(* Logix 5000 project; controller Drives_Line1 1756-L72 rev 20.13; software revision 20.04; part 14 of 21 *)
(* tags used below, declared in another part *)
   zEntry_Accu_MaxAccDec : REAL;
   zEntry_Accu_SpdRegMax : REAL;
   zEntry_Accu_SpdRegMin : REAL;
   Bridle_01 : UDT_Bridle_3M;
   Bridle_02 : UDT_Bridle_2M;
   Bridle_03 : UDT_Bridle_2M;
   Entry_Accu : UDT_Entry_Accu;
   EntryCtrl : UDT_Control_Zone;
   In_Commands : UDT_Commands;
   In_Config : UDT_Config;
   In_Setpoints : UDT_Setpoints;
   LineCmd : UDT_Commands_Line;
   LineCtrl : UDT_Control_Line;
   Out_Feedbacks : UDT_Fdbks;
   Out_Status : UDT_Status;
   TestConfig_Entry_Accu : UDT_Config_Accu;
   TM1 : UDT_TM;
   TM2 : UDT_TM;
   zConfigFromMaster : BOOL;
   zExit_Accu_NrOfCyl : DINT;
(* P16_Entry_Accu, continued *)

ROUTINE R12_DriveRef   (* function block diagram *)
   SHEET 1   // Speed reference selection
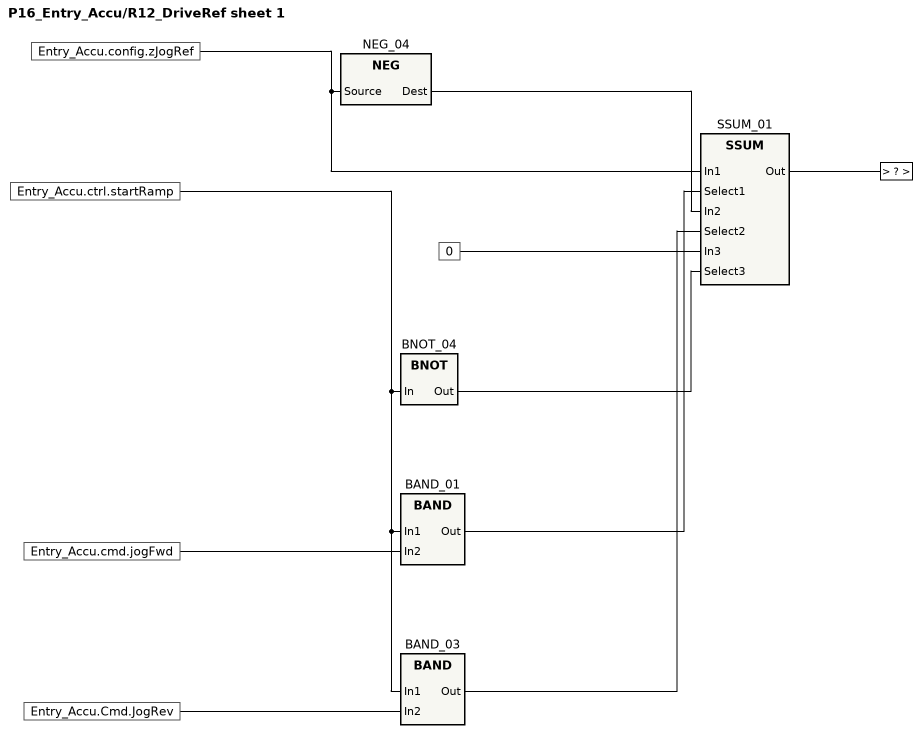
   NEG_04 : NEG(Source := Entry_Accu.config.zJogRef);
   BNOT_04 : BNOT(In := Entry_Accu.ctrl.startRamp);
   BAND_01 : BAND(In1 := Entry_Accu.ctrl.startRamp, In2 := Entry_Accu.cmd.jogFwd);
   BAND_03 : BAND(In1 := Entry_Accu.ctrl.startRamp, In2 := Entry_Accu.Cmd.JogRev);
   SSUM_01 : SSUM(In1 := Entry_Accu.config.zJogRef, Select1 := BAND_01.Out, In2 := NEG_04.Dest, Select2 := BAND_03.Out, In3 := 0, Select3 := BNOT_04.Out);
   WIRE(?) := SSUM_01.Out;
   SHEET 2   // S-Curve
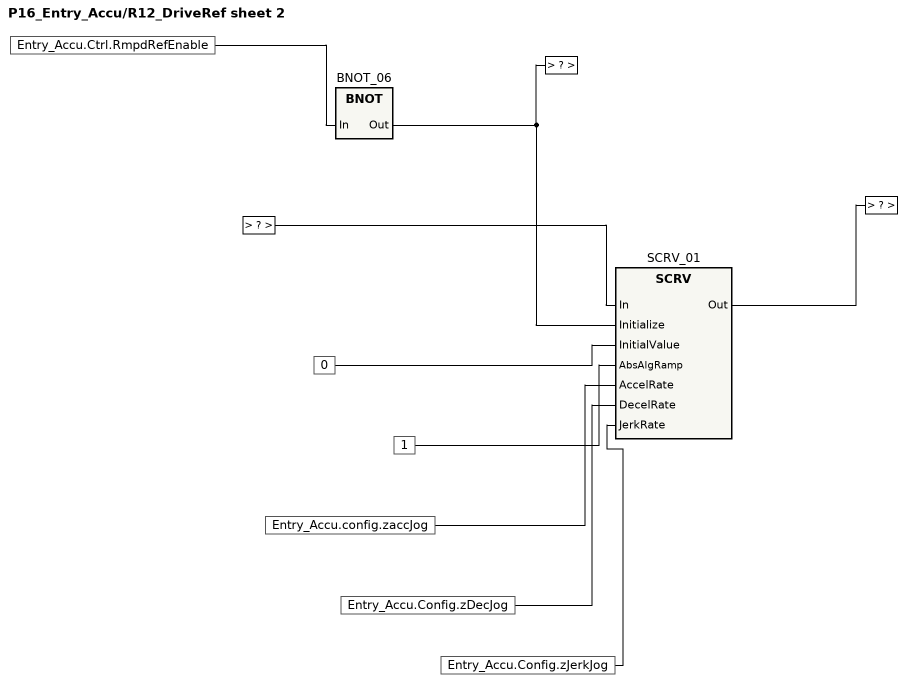
   BNOT_06 : BNOT(In := Entry_Accu.Ctrl.RmpdRefEnable);
   WIRE(?) := BNOT_06.Out;
   SCRV_01 : SCRV(In := WIRE(?), Initialize := BNOT_06.Out, InitialValue := 0, AbsAlgRamp := 1, AccelRate := Entry_Accu.config.zaccJog, DecelRate := Entry_Accu.Config.zDecJog, JerkRate := Entry_Accu.Config.zJerkJog);
   WIRE(?) := SCRV_01.Out;
   SHEET 3   // Run speed reference (Ve - Vp)
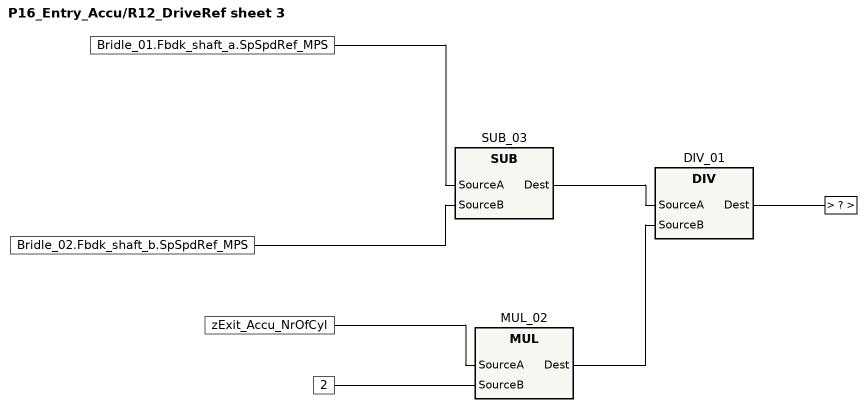
   SUB_03 : SUB(SourceA := Bridle_01.Fbdk_shaft_a.SpSpdRef_MPS, SourceB := Bridle_02.Fbdk_shaft_b.SpSpdRef_MPS);
   MUL_02 : MUL(SourceA := zExit_Accu_NrOfCyl, SourceB := 2);
   DIV_01 : DIV(SourceA := SUB_03.Dest, SourceB := MUL_02.Dest);
   WIRE(?) := DIV_01.Dest;
   SHEET 4   // Select ramped/unramped reference
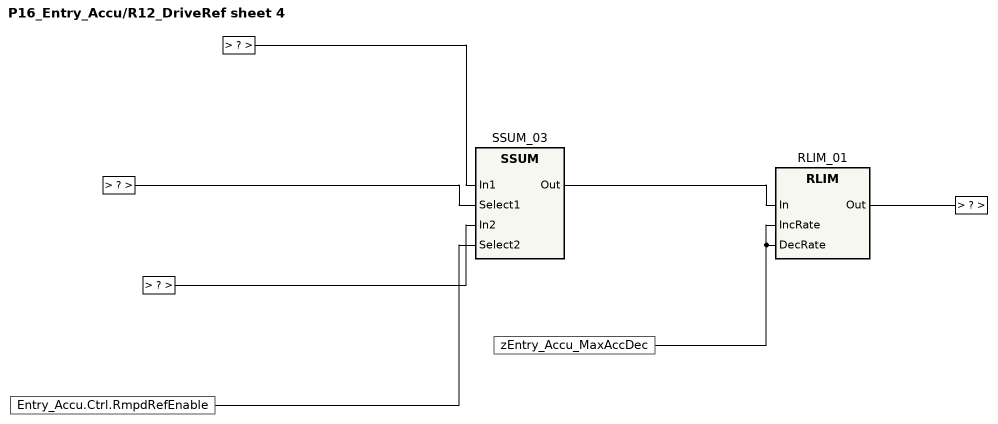
   SSUM_03 : SSUM(In1 := WIRE(?), Select1 := WIRE(?), In2 := WIRE(?), Select2 := Entry_Accu.Ctrl.RmpdRefEnable);
   RLIM_01 : RLIM(In := SSUM_03.Out, IncRate := zEntry_Accu_MaxAccDec, DecRate := zEntry_Accu_MaxAccDec);
   WIRE(?) := RLIM_01.Out;
   SHEET 5   // Speed regulator limits
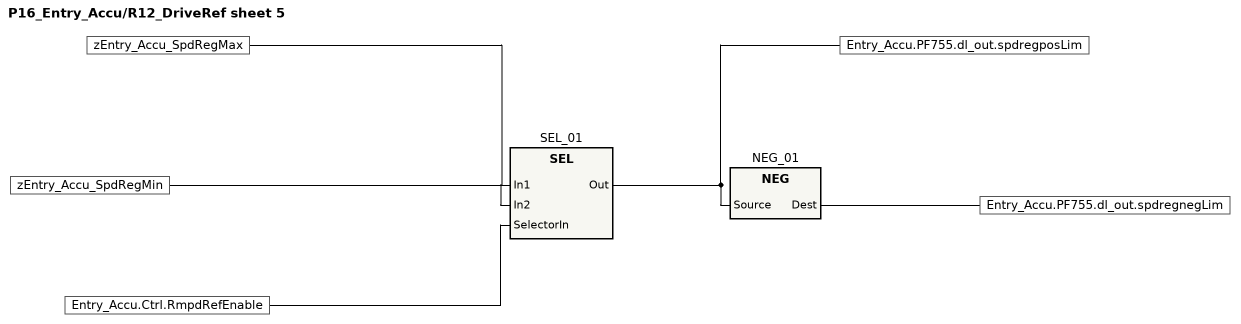
   SEL_01 : SEL(In1 := zEntry_Accu_SpdRegMax, In2 := zEntry_Accu_SpdRegMin, SelectorIn := Entry_Accu.Ctrl.RmpdRefEnable);
   NEG_01 : NEG(Source := SEL_01.Out);
   Entry_Accu.PF755.dl_out.spdregposLim := SEL_01.Out;
   Entry_Accu.PF755.dl_out.spdregnegLim := NEG_01.Dest;
   SHEET 6   // Final speed reference
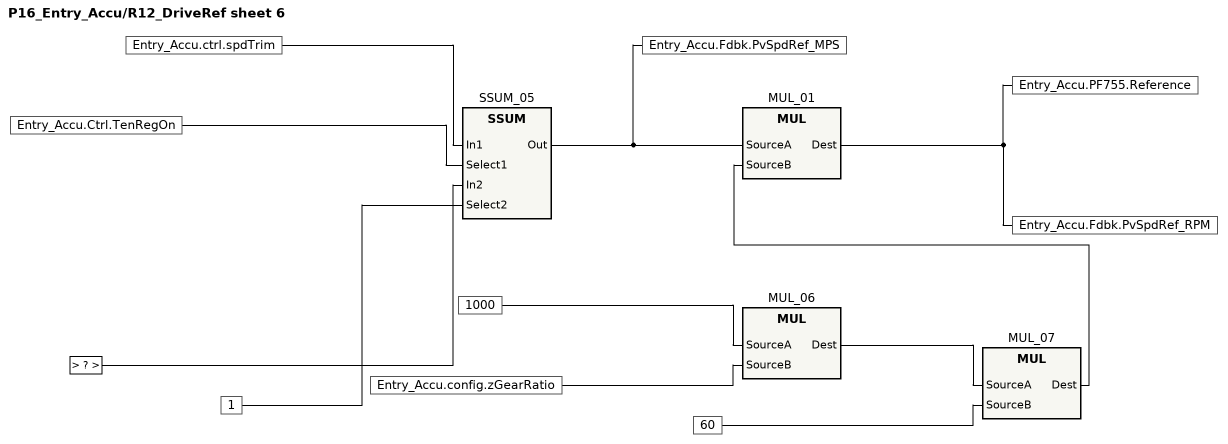
   SSUM_05 : SSUM(In1 := Entry_Accu.ctrl.spdTrim, Select1 := Entry_Accu.Ctrl.TenRegOn, In2 := WIRE(?), Select2 := 1);
   Entry_Accu.Fdbk.PvSpdRef_MPS := SSUM_05.Out;
   MUL_06 : MUL(SourceA := 1000, SourceB := Entry_Accu.config.zGearRatio);
   MUL_07 : MUL(SourceA := MUL_06.Dest, SourceB := 60);
   MUL_01 : MUL(SourceA := SSUM_05.Out, SourceB := MUL_07.Dest);
   Entry_Accu.PF755.Reference := MUL_01.Dest;
   Entry_Accu.Fdbk.PvSpdRef_RPM := MUL_01.Dest;
END_ROUTINE

ROUTINE R98_ToDrive   (* ladder *)
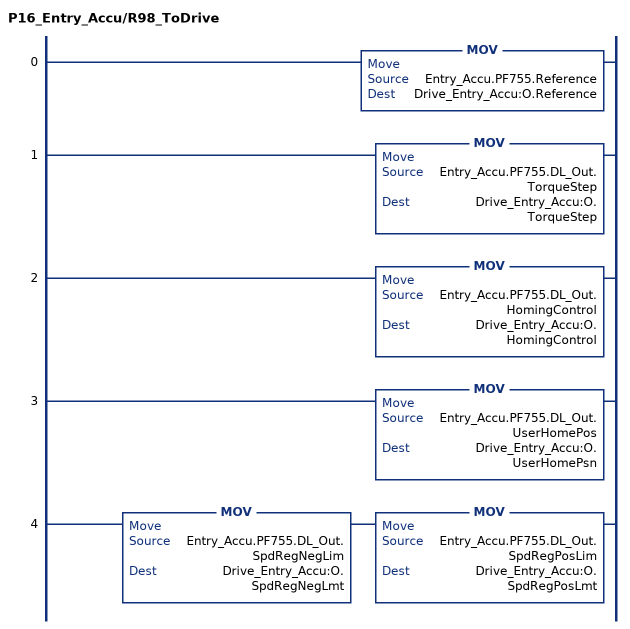
   0: MOV(Entry_Accu.PF755.Reference,Drive_Entry_Accu:O.Reference);
   1: MOV(Entry_Accu.PF755.DL_Out.TorqueStep,Drive_Entry_Accu:O.TorqueStep);
   2: MOV(Entry_Accu.PF755.DL_Out.HomingControl,Drive_Entry_Accu:O.HomingControl);
   3: MOV(Entry_Accu.PF755.DL_Out.UserHomePos,Drive_Entry_Accu:O.UserHomePsn);
   4: MOV(Entry_Accu.PF755.DL_Out.SpdRegNegLim,Drive_Entry_Accu:O.SpdRegNegLmt)MOV(Entry_Accu.PF755.DL_Out.SpdRegPosLim,Drive_Entry_Accu:O.SpdRegPosLmt);
END_ROUTINE

ROUTINE R999_Test   (* ladder *)
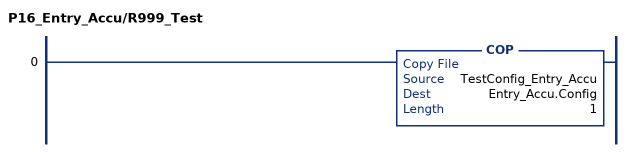
   0: COP(TestConfig_Entry_Accu,Entry_Accu.Config,1);
END_ROUTINE

ROUTINE R99_To_Master   (* ladder *)
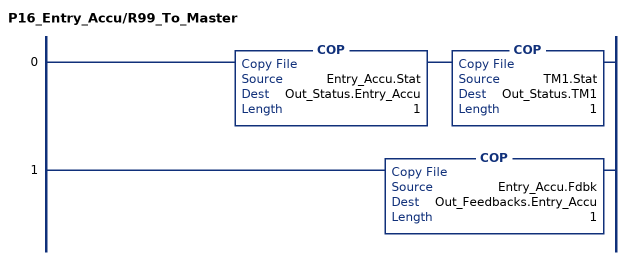
   0: COP(Entry_Accu.Stat,Out_Status.Entry_Accu,1)COP(TM1.Stat,Out_Status.TM1,1);
   1: COP(Entry_Accu.Fdbk,Out_Feedbacks.Entry_Accu,1);
END_ROUTINE
END_PROGRAM

PROGRAM P17_Bridle_03   (* main routine R00_Main *)
VAR
   ABS_01 : FBD_MATH_ADVANCED := (Source := 0.00068994303, Dest := 0.00068994303);
   ADD_01 : FBD_MATH := (SourceA := 0.00068994303, Dest := 0.00068994303);
   BAND_01 : FBD_BOOLEAN_AND := (In3 := 1, In4 := 1, In5 := 1, In6 := 1, In7 := 1, In8 := 1);
   BAND_03 : FBD_BOOLEAN_AND := (In3 := 1, In4 := 1, In5 := 1, In6 := 1, In7 := 1, In8 := 1);
   BNOT_01 : FBD_BOOLEAN_NOT := (Out := 1);
   BNOT_02 : FBD_BOOLEAN_NOT := (Out := 1);
   BNOT_04 : FBD_BOOLEAN_NOT := (Out := 1);
   BNOT_06 : FBD_BOOLEAN_NOT := (Out := 1);
   BOR_01 : FBD_BOOLEAN_OR;
   Bridle_03_Rev_mm : REAL := 0.10188699;
   Bridle_03_SpdTrimMPS : REAL;
   Bridle_03_SpdTrimPct : REAL;
   Bridle_03a_FBCounts_mm : REAL := 417.3291;
   Bridle_03a_RPMPerMPS : REAL := 6113.219;
   Bridle_03b_RPMPerMPS : REAL := 6113.219;
   DIV_01 : FBD_MATH := (SourceB := 100.0);
   DIV_03 : FBD_MATH := (SourceA := 1.523458, SourceB := 100.0, Dest := 0.01523458);
   EQU_01 : FBD_COMPARE := (SourceA := 0.08463864);
   IO_State_Bridle_03a : INT := 4;
   IO_State_Bridle_03b : INT := 4;
   IO_State_Tmp_Bridle_03a : INT := 16384;
   IO_State_Tmp_Bridle_03b : INT := 16384;
   MUL_01 : FBD_MATH := (SourceA := 0.00068994303, SourceB := 6113.219, Dest := 4.217773);
   MUL_02 : FBD_MATH := (SourceA := 6113.219, SourceB := 0.00068994303, Dest := 4.217773);
   MUL_04 : FBD_MATH := (SourceB := 0.25);
   MUL_05 : FBD_MATH := (SourceB := 0.00068994303);
   NEG_03 : FBD_MATH_ADVANCED := (Source := 0.01523458, Dest := -0.01523458);
   NEG_04 : FBD_MATH_ADVANCED := (Source := 0.083, Dest := -0.083);
   Ons : DINT;
   PI_02 : PROP_INT := (In := -2.3841858e-07, Initialize := 1, Kp := 0.15, Wld := 0.1, HighLimit := 2.5, LowLimit := -2.5, ShapeKpPlus := 1.0, ShapeKpMinus := 1.0, ShapeWldPlus := 1.0, ShapeWldMinus := 1.0, RTSTime := 1, DeltaT := 0.05);
   PI_03 : PROP_INT := (In := 0.1284, Initialize := 1, Kp := 0.15, Wld := 0.08, HighLimit := 0.01523458, LowLimit := -0.01523458, ShapeKpPlus := 1.0, ShapeKpMinus := 1.0, ShapeWldPlus := 1.0, ShapeWldMinus := 1.0, RTSTime := 1, DeltaT := 0.05);
   PulsReset_PID : TIMER := (PRE := 250);
   RLIM_01 : RATE_LIMITER := (In := 0.00068994303, IncRate := 0.25, DecRate := 0.25, RTSTime := 1, Out := 0.00068994303, DeltaT := 0.05);
   SCL_01 : SCALE := (In := 0.00068994303, InRawMax := 0.25, InEUMax := 10.0, InEUMin := 1.5, Limiting := 1, Out := 1.523458);
   SCL_04 : SCALE := (In := 8250.0, InRawMax := 50000.0, InEUMax := 1.0, Limiting := 1, Out := 0.16499999);
   SCL_05 : SCALE := (In := 1820.0, InRawMax := 50000.0, InEUMax := 1.0, Limiting := 1, Out := 0.036399998);
   SCL_09 : SCALE := (InRawMax := 100.0, InRawMin := -100.0, InEUMax := 2.5, InEUMin := -2.5, Limiting := 1, Out := -2.3841858e-07);
   SCRV_01 : S_CURVE := (Initialize := 1, AbsAlgRamp := 1, AccelRate := 0.083, DecelRate := 0.083, JerkRate := 0.1, RTSTime := 1, DeltaT := 0.05);
   SSUM_05 : SELECTED_SUMMER := (In1 := 0.083, Gain1 := 1.0, In2 := -0.083, Gain2 := 1.0, Gain3 := 1.0, Select3 := 1, Gain4 := 1.0, Gain5 := 1.0, Gain6 := 1.0, Gain7 := 1.0, Gain8 := 1.0);
   SSUM_07 : SELECTED_SUMMER := (In1 := 0.00068994303, Gain1 := 1.0, Select1 := 1, Gain2 := 1.0, Gain3 := 1.0, Gain4 := 1.0, Gain5 := 1.0, Gain6 := 1.0, Gain7 := 1.0, Gain8 := 1.0, Out := 0.00068994303);
   SSUM_09 : SELECTED_SUMMER := (In1 := 0.00068994303, Gain1 := 1.0, Select1 := 1, Gain2 := 1.0, Gain3 := 1.0, Gain4 := 1.0, Gain5 := 1.0, Gain6 := 1.0, Gain7 := 1.0, Gain8 := 1.0, Out := 0.00068994303);
   SUB_02 : FBD_MATH;
   SUB_03 : FBD_MATH := (SourceA := 0.16499999, SourceB := 0.0372, Dest := 0.12779999);
   TimeOn_PIDOn : TIMER := (PRE := 500);
   TofReset : TIMER := (PRE := 1000, ACC := 1000);
   TonNoResponse : TIMER[3] := ([0].PRE := 2500, [1].PRE := 2500, [2].PRE := 2500, [2].ACC := 2500, [2].EN := 1, [2].DN := 1);
   TonRefOn : TIMER := (PRE := 500);
   TonTensionOnSp : TIMER := (PRE := 500);
   zBridle_03_EncRes : DINT := 4096;
   zBridle_03_Ki_SpdTrim : REAL := 0.1;
   zBridle_03_Kp_SpdTrim : REAL := 0.15;
   zBridle_03_Kp_Treg : REAL := 0.15;
   zBridle_03_MaxAccDec : REAL := 0.25;
   zBridle_03_MaxTrimSpdTrim : REAL := 2.5;
   zBridle_03_MinTrimSpdTrim : REAL := -2.5;
   zBridle_03_Trim_HL : REAL := 10.0;
   zBridle_03_Trim_LL : REAL := 1.5;
   zBridle_03_WLD_Treg : REAL := 0.08;
   zTM2_Tens_Offset : REAL := 200.0;
END_VAR

ROUTINE R00_Main   (* ladder *)
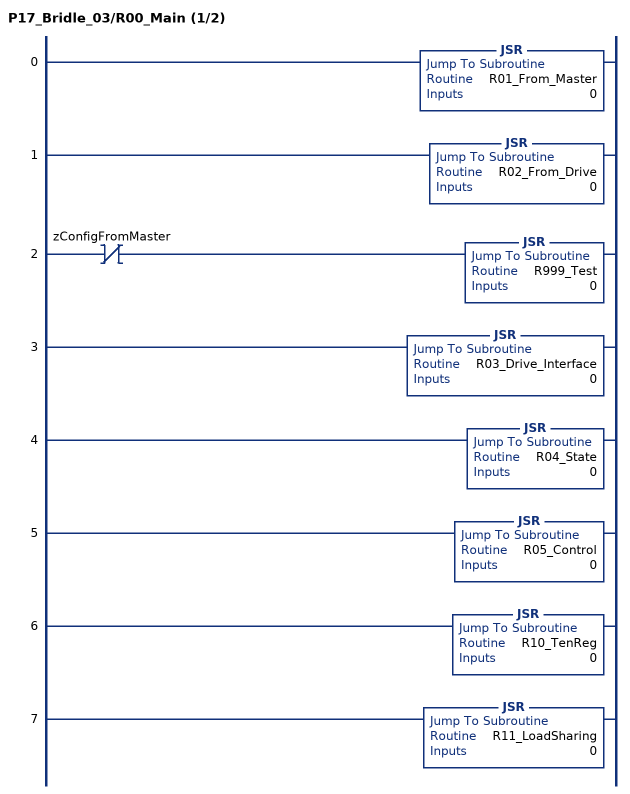
   0: JSR(R01_From_Master,0);
   1: JSR(R02_From_Drive,0);
   2: XIO(zConfigFromMaster)JSR(R999_Test,0);
   3: JSR(R03_Drive_Interface,0);
   4: JSR(R04_State,0);
   5: JSR(R05_Control,0);
   6: JSR(R10_TenReg,0);
   7: JSR(R11_LoadSharing,0);
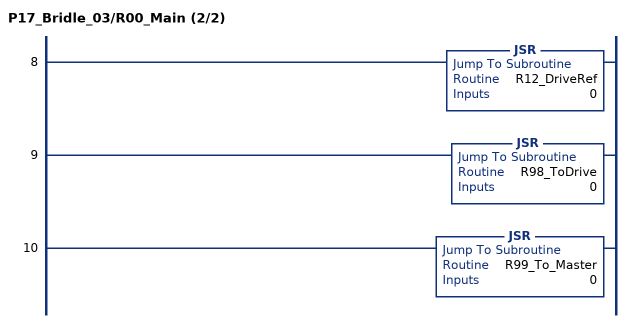
   8: JSR(R12_DriveRef,0);
   9: JSR(R98_ToDrive,0);
   10: JSR(R99_To_Master,0);
END_ROUTINE

ROUTINE R01_From_Master   (* ladder *)
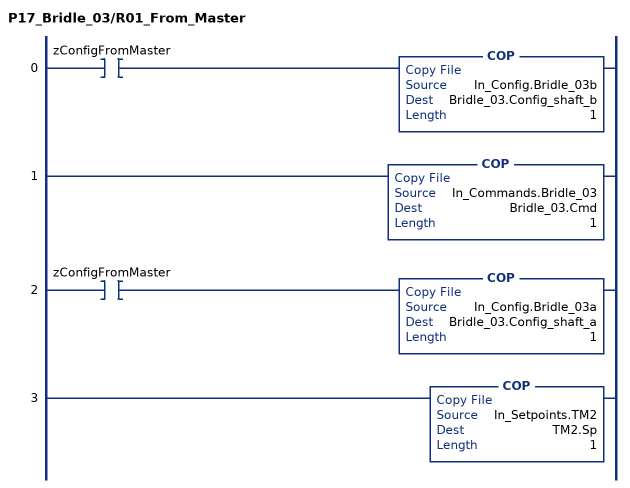
   0: XIC(zConfigFromMaster)COP(In_Config.Bridle_03b,Bridle_03.Config_shaft_b,1);
   1: COP(In_Commands.Bridle_03,Bridle_03.Cmd,1);
   2: XIC(zConfigFromMaster)COP(In_Config.Bridle_03a,Bridle_03.Config_shaft_a,1);
   3: COP(In_Setpoints.TM2,TM2.Sp,1);
END_ROUTINE

ROUTINE R02_From_Drive   (* ladder *)
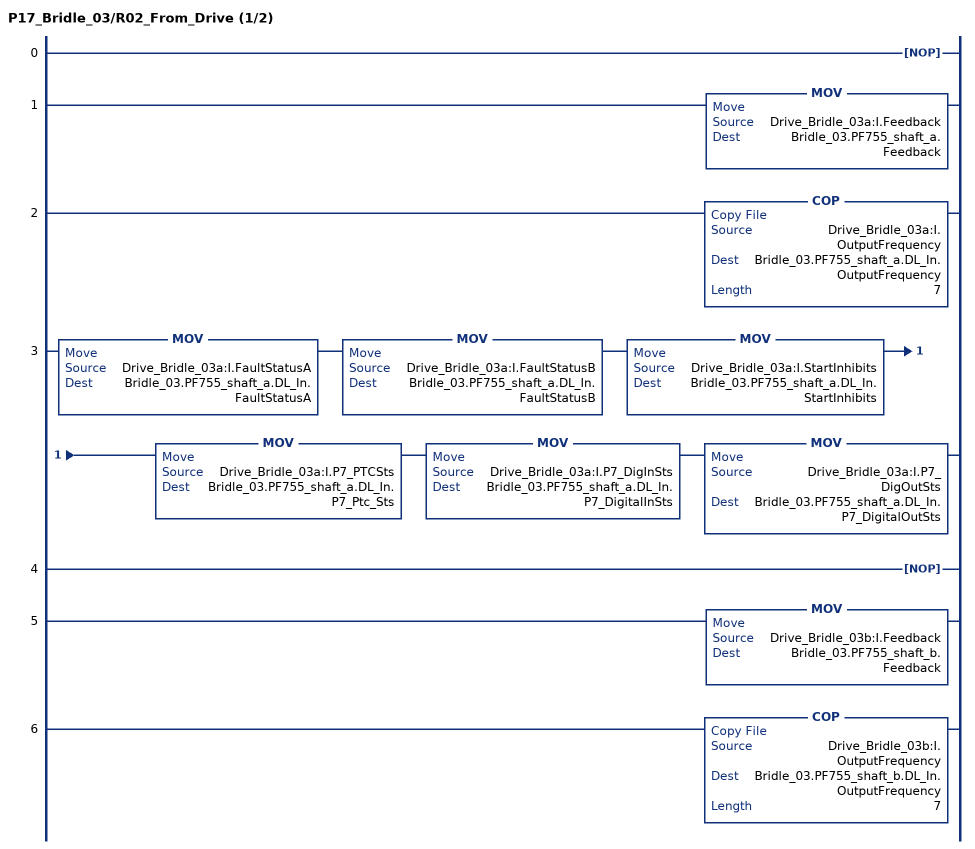
   0: NOP();
   1: MOV(Drive_Bridle_03a:I.Feedback,Bridle_03.PF755_shaft_a.Feedback);
   2: COP(Drive_Bridle_03a:I.OutputFrequency,Bridle_03.PF755_shaft_a.DL_In.OutputFrequency,7);
   3: MOV(Drive_Bridle_03a:I.FaultStatusA,Bridle_03.PF755_shaft_a.DL_In.FaultStatusA)MOV(Drive_Bridle_03a:I.FaultStatusB,Bridle_03.PF755_shaft_a.DL_In.FaultStatusB)MOV(Drive_Bridle_03a:I.StartInhibits,Bridle_03.PF755_shaft_a.DL_In.StartInhibits)MOV(Drive_Bridle_03a:I.P7_PTCSts,Bridle_03.PF755_shaft_a.DL_In.P7_Ptc_Sts)MOV(Drive_Bridle_03a:I.P7_DigInSts,Bridle_03.PF755_shaft_a.DL_In.P7_DigitalInSts)MOV(Drive_Bridle_03a:I.P7_DigOutSts,Bridle_03.PF755_shaft_a.DL_In.P7_DigitalOutSts);
   4: NOP();
   5: MOV(Drive_Bridle_03b:I.Feedback,Bridle_03.PF755_shaft_b.Feedback);
   6: COP(Drive_Bridle_03b:I.OutputFrequency,Bridle_03.PF755_shaft_b.DL_In.OutputFrequency,7);
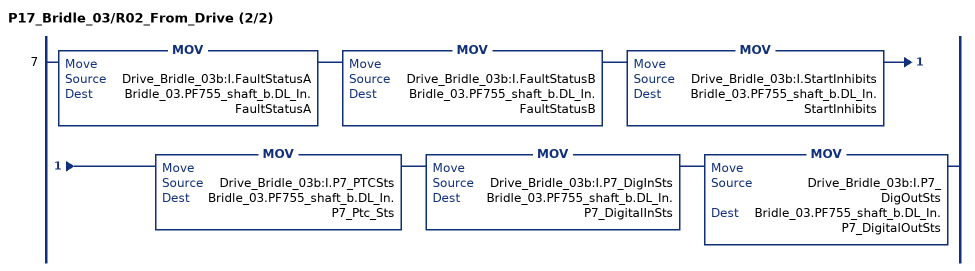
   7: MOV(Drive_Bridle_03b:I.FaultStatusA,Bridle_03.PF755_shaft_b.DL_In.FaultStatusA)MOV(Drive_Bridle_03b:I.FaultStatusB,Bridle_03.PF755_shaft_b.DL_In.FaultStatusB)MOV(Drive_Bridle_03b:I.StartInhibits,Bridle_03.PF755_shaft_b.DL_In.StartInhibits)MOV(Drive_Bridle_03b:I.P7_PTCSts,Bridle_03.PF755_shaft_b.DL_In.P7_Ptc_Sts)MOV(Drive_Bridle_03b:I.P7_DigInSts,Bridle_03.PF755_shaft_b.DL_In.P7_DigitalInSts)MOV(Drive_Bridle_03b:I.P7_DigOutSts,Bridle_03.PF755_shaft_b.DL_In.P7_DigitalOutSts);
END_ROUTINE

ROUTINE R03_Drive_Interface   (* ladder *)
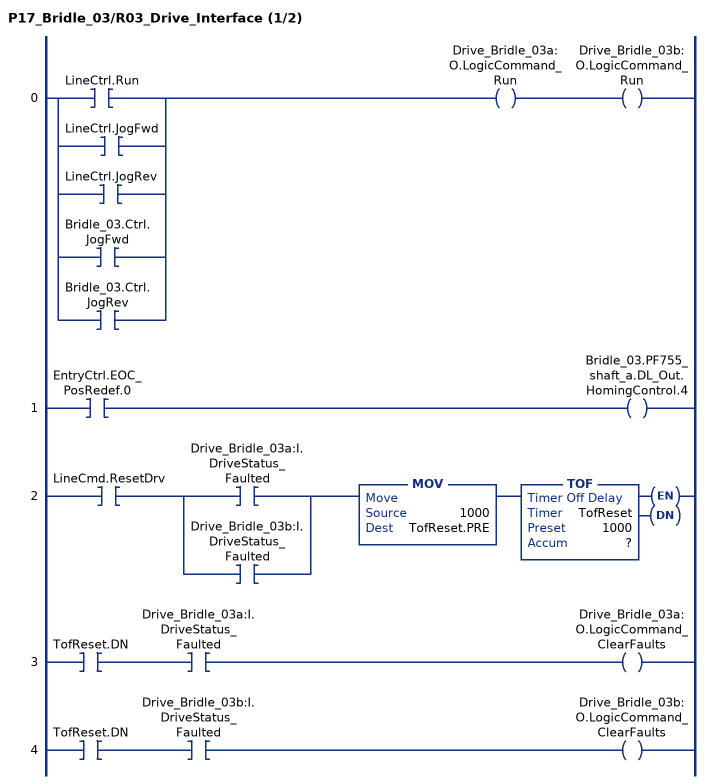
   0: [XIC(LineCtrl.Run) ,XIC(LineCtrl.JogFwd) ,XIC(LineCtrl.JogRev) ,XIC(Bridle_03.Ctrl.JogFwd) ,XIC(Bridle_03.Ctrl.JogRev) ]OTE(Drive_Bridle_03a:O.LogicCommand_Run)OTE(Drive_Bridle_03b:O.LogicCommand_Run);
   1: XIC(EntryCtrl.EOC_PosRedef.0)OTE(Bridle_03.PF755_shaft_a.DL_Out.HomingControl.4);
   2: XIC(LineCmd.ResetDrv)[XIC(Drive_Bridle_03a:I.DriveStatus_Faulted) ,XIC(Drive_Bridle_03b:I.DriveStatus_Faulted) ]MOV(1000,TofReset.PRE)TOF(TofReset,?,?);
   3: XIC(TofReset.DN)XIC(Drive_Bridle_03a:I.DriveStatus_Faulted)OTE(Drive_Bridle_03a:O.LogicCommand_ClearFaults);
   4: XIC(TofReset.DN)XIC(Drive_Bridle_03b:I.DriveStatus_Faulted)OTE(Drive_Bridle_03b:O.LogicCommand_ClearFaults);
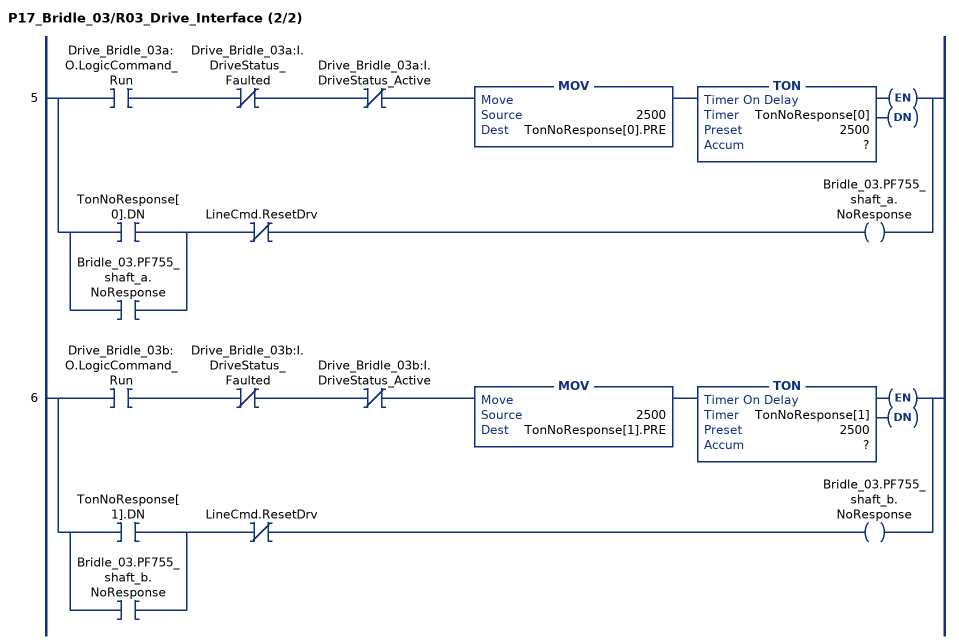
   5: [XIC(Drive_Bridle_03a:O.LogicCommand_Run) XIO(Drive_Bridle_03a:I.DriveStatus_Faulted) XIO(Drive_Bridle_03a:I.DriveStatus_Active) MOV(2500,TonNoResponse[0].PRE) TON(TonNoResponse[0],?,?) ,[XIC(TonNoResponse[0].DN) ,XIC(Bridle_03.PF755_shaft_a.NoResponse) ] XIO(LineCmd.ResetDrv) OTE(Bridle_03.PF755_shaft_a.NoResponse) ];
   6: [XIC(Drive_Bridle_03b:O.LogicCommand_Run) XIO(Drive_Bridle_03b:I.DriveStatus_Faulted) XIO(Drive_Bridle_03b:I.DriveStatus_Active) MOV(2500,TonNoResponse[1].PRE) TON(TonNoResponse[1],?,?) ,[XIC(TonNoResponse[1].DN) ,XIC(Bridle_03.PF755_shaft_b.NoResponse) ] XIO(LineCmd.ResetDrv) OTE(Bridle_03.PF755_shaft_b.NoResponse) ];
END_ROUTINE

ROUTINE R04_State   (* ladder *)
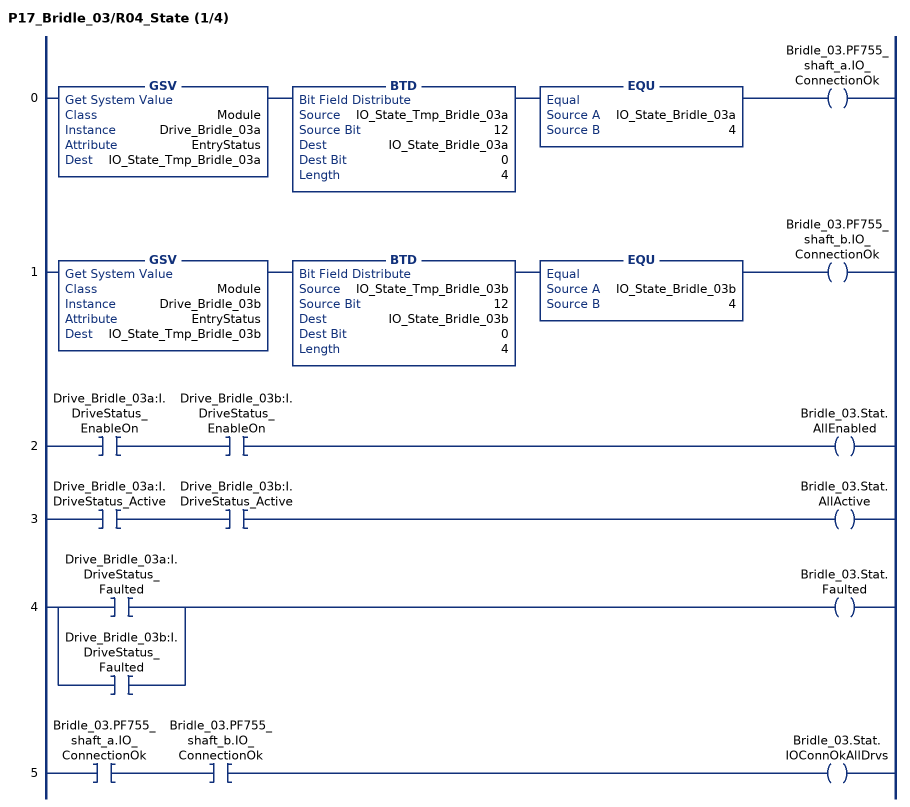
   0: GSV(Module,Drive_Bridle_03a,EntryStatus,IO_State_Tmp_Bridle_03a)BTD(IO_State_Tmp_Bridle_03a,12,IO_State_Bridle_03a,0,4)EQU(IO_State_Bridle_03a,4)OTE(Bridle_03.PF755_shaft_a.IO_ConnectionOk);
   1: GSV(Module,Drive_Bridle_03b,EntryStatus,IO_State_Tmp_Bridle_03b)BTD(IO_State_Tmp_Bridle_03b,12,IO_State_Bridle_03b,0,4)EQU(IO_State_Bridle_03b,4)OTE(Bridle_03.PF755_shaft_b.IO_ConnectionOk);
   2: XIC(Drive_Bridle_03a:I.DriveStatus_EnableOn)XIC(Drive_Bridle_03b:I.DriveStatus_EnableOn)OTE(Bridle_03.Stat.AllEnabled);
   3: XIC(Drive_Bridle_03a:I.DriveStatus_Active)XIC(Drive_Bridle_03b:I.DriveStatus_Active)OTE(Bridle_03.Stat.AllActive);
   4: [XIC(Drive_Bridle_03a:I.DriveStatus_Faulted) ,XIC(Drive_Bridle_03b:I.DriveStatus_Faulted) ]OTE(Bridle_03.Stat.Faulted);
   5: XIC(Bridle_03.PF755_shaft_a.IO_ConnectionOk)XIC(Bridle_03.PF755_shaft_b.IO_ConnectionOk)OTE(Bridle_03.Stat.IOConnOkAllDrvs);
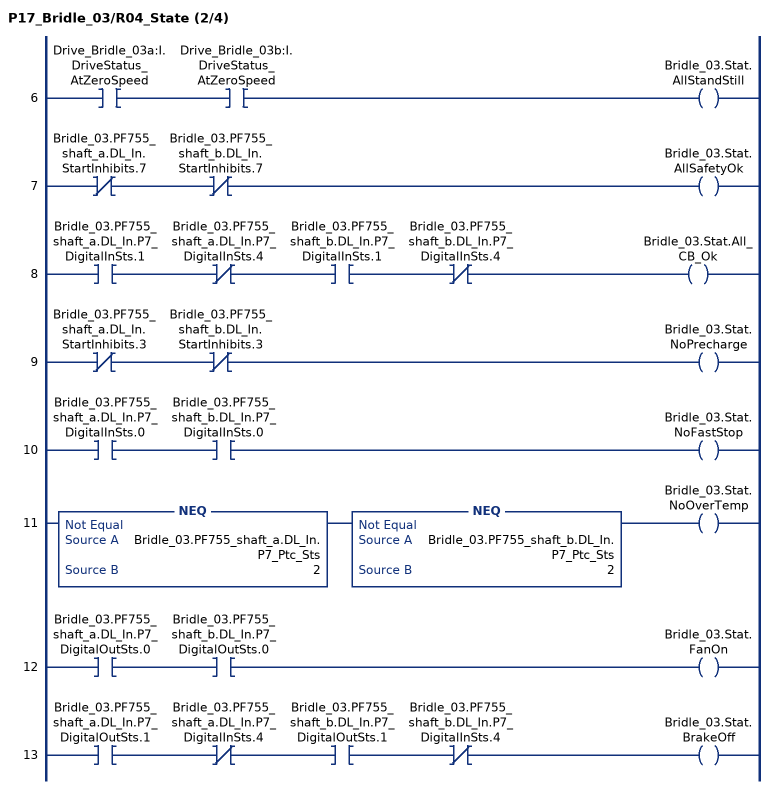
   6: XIC(Drive_Bridle_03a:I.DriveStatus_AtZeroSpeed)XIC(Drive_Bridle_03b:I.DriveStatus_AtZeroSpeed)OTE(Bridle_03.Stat.AllStandStill);
   7: XIO(Bridle_03.PF755_shaft_a.DL_In.StartInhibits.7)XIO(Bridle_03.PF755_shaft_b.DL_In.StartInhibits.7)OTE(Bridle_03.Stat.AllSafetyOk);
   8: XIC(Bridle_03.PF755_shaft_a.DL_In.P7_DigitalInSts.1)XIO(Bridle_03.PF755_shaft_a.DL_In.P7_DigitalInSts.4)XIC(Bridle_03.PF755_shaft_b.DL_In.P7_DigitalInSts.1)XIO(Bridle_03.PF755_shaft_b.DL_In.P7_DigitalInSts.4)OTE(Bridle_03.Stat.All_CB_Ok);
   9: XIO(Bridle_03.PF755_shaft_a.DL_In.StartInhibits.3)XIO(Bridle_03.PF755_shaft_b.DL_In.StartInhibits.3)OTE(Bridle_03.Stat.NoPrecharge);
   10: XIC(Bridle_03.PF755_shaft_a.DL_In.P7_DigitalInSts.0)XIC(Bridle_03.PF755_shaft_b.DL_In.P7_DigitalInSts.0)OTE(Bridle_03.Stat.NoFastStop);
   11: NEQ(Bridle_03.PF755_shaft_a.DL_In.P7_Ptc_Sts,2)NEQ(Bridle_03.PF755_shaft_b.DL_In.P7_Ptc_Sts,2)OTE(Bridle_03.Stat.NoOverTemp);
   12: XIC(Bridle_03.PF755_shaft_a.DL_In.P7_DigitalOutSts.0)XIC(Bridle_03.PF755_shaft_b.DL_In.P7_DigitalOutSts.0)OTE(Bridle_03.Stat.FanOn);
   13: XIC(Bridle_03.PF755_shaft_a.DL_In.P7_DigitalOutSts.1)XIO(Bridle_03.PF755_shaft_a.DL_In.P7_DigitalInSts.4)XIC(Bridle_03.PF755_shaft_b.DL_In.P7_DigitalOutSts.1)XIO(Bridle_03.PF755_shaft_b.DL_In.P7_DigitalInSts.4)OTE(Bridle_03.Stat.BrakeOff);
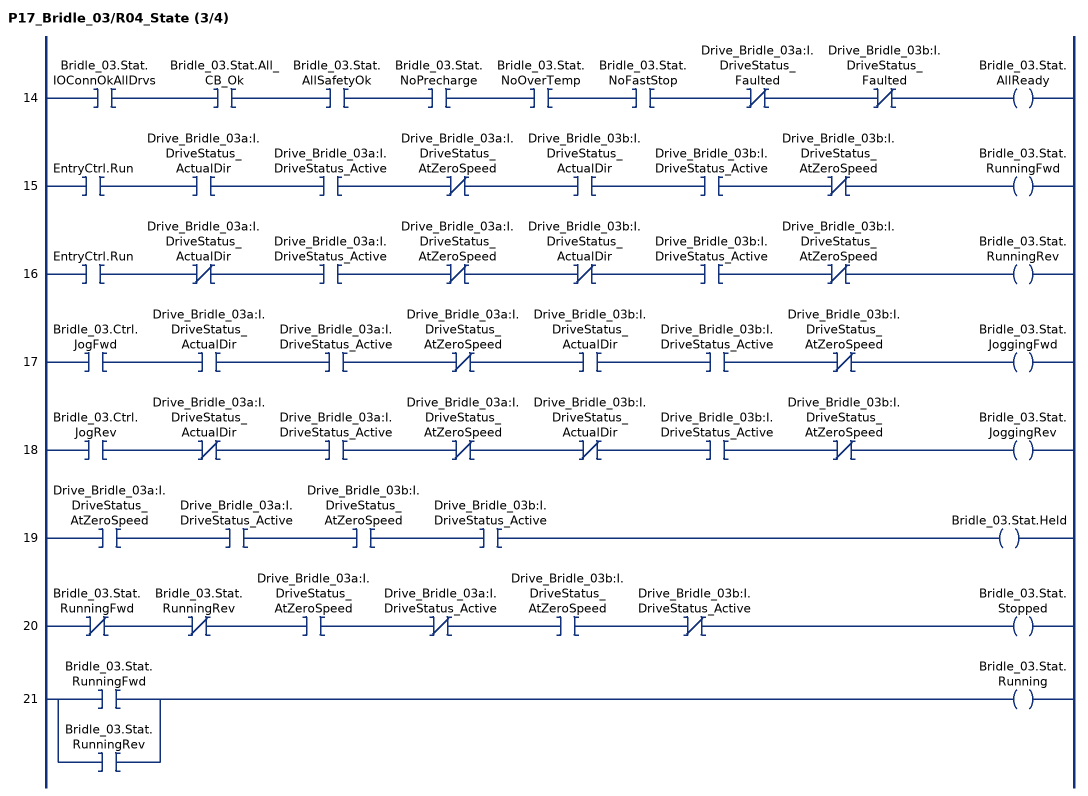
   14: XIC(Bridle_03.Stat.IOConnOkAllDrvs)XIC(Bridle_03.Stat.All_CB_Ok)XIC(Bridle_03.Stat.AllSafetyOk)XIC(Bridle_03.Stat.NoPrecharge)XIC(Bridle_03.Stat.NoOverTemp)XIC(Bridle_03.Stat.NoFastStop)XIO(Drive_Bridle_03a:I.DriveStatus_Faulted)XIO(Drive_Bridle_03b:I.DriveStatus_Faulted)OTE(Bridle_03.Stat.AllReady);
   15: XIC(EntryCtrl.Run)XIC(Drive_Bridle_03a:I.DriveStatus_ActualDir)XIC(Drive_Bridle_03a:I.DriveStatus_Active)XIO(Drive_Bridle_03a:I.DriveStatus_AtZeroSpeed)XIC(Drive_Bridle_03b:I.DriveStatus_ActualDir)XIC(Drive_Bridle_03b:I.DriveStatus_Active)XIO(Drive_Bridle_03b:I.DriveStatus_AtZeroSpeed)OTE(Bridle_03.Stat.RunningFwd);
   16: XIC(EntryCtrl.Run)XIO(Drive_Bridle_03a:I.DriveStatus_ActualDir)XIC(Drive_Bridle_03a:I.DriveStatus_Active)XIO(Drive_Bridle_03a:I.DriveStatus_AtZeroSpeed)XIO(Drive_Bridle_03b:I.DriveStatus_ActualDir)XIC(Drive_Bridle_03b:I.DriveStatus_Active)XIO(Drive_Bridle_03b:I.DriveStatus_AtZeroSpeed)OTE(Bridle_03.Stat.RunningRev);
   17: XIC(Bridle_03.Ctrl.JogFwd)XIC(Drive_Bridle_03a:I.DriveStatus_ActualDir)XIC(Drive_Bridle_03a:I.DriveStatus_Active)XIO(Drive_Bridle_03a:I.DriveStatus_AtZeroSpeed)XIC(Drive_Bridle_03b:I.DriveStatus_ActualDir)XIC(Drive_Bridle_03b:I.DriveStatus_Active)XIO(Drive_Bridle_03b:I.DriveStatus_AtZeroSpeed)OTE(Bridle_03.Stat.JoggingFwd);
   18: XIC(Bridle_03.Ctrl.JogRev)XIO(Drive_Bridle_03a:I.DriveStatus_ActualDir)XIC(Drive_Bridle_03a:I.DriveStatus_Active)XIO(Drive_Bridle_03a:I.DriveStatus_AtZeroSpeed)XIO(Drive_Bridle_03b:I.DriveStatus_ActualDir)XIC(Drive_Bridle_03b:I.DriveStatus_Active)XIO(Drive_Bridle_03b:I.DriveStatus_AtZeroSpeed)OTE(Bridle_03.Stat.JoggingRev);
   19: XIC(Drive_Bridle_03a:I.DriveStatus_AtZeroSpeed)XIC(Drive_Bridle_03a:I.DriveStatus_Active)XIC(Drive_Bridle_03b:I.DriveStatus_AtZeroSpeed)XIC(Drive_Bridle_03b:I.DriveStatus_Active)OTE(Bridle_03.Stat.Held);
   20: XIO(Bridle_03.Stat.RunningFwd)XIO(Bridle_03.Stat.RunningRev)XIC(Drive_Bridle_03a:I.DriveStatus_AtZeroSpeed)XIO(Drive_Bridle_03a:I.DriveStatus_Active)XIC(Drive_Bridle_03b:I.DriveStatus_AtZeroSpeed)XIO(Drive_Bridle_03b:I.DriveStatus_Active)OTE(Bridle_03.Stat.Stopped);
   21: [XIC(Bridle_03.Stat.RunningFwd) ,XIC(Bridle_03.Stat.RunningRev) ]OTE(Bridle_03.Stat.Running);
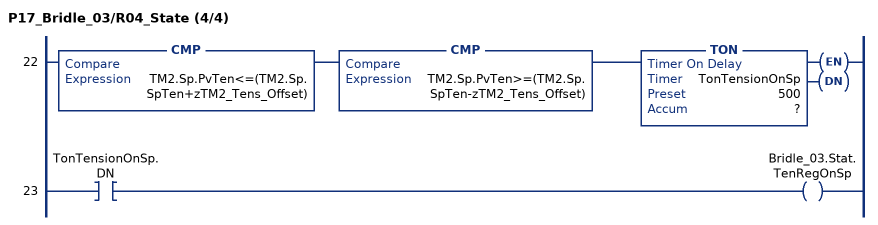
   22: CMP(TM2.Sp.PvTen<=(TM2.Sp.SpTen+zTM2_Tens_Offset))CMP(TM2.Sp.PvTen>=(TM2.Sp.SpTen-zTM2_Tens_Offset))TON(TonTensionOnSp,?,?);
   23: XIC(TonTensionOnSp.DN)OTE(Bridle_03.Stat.TenRegOnSp);
END_ROUTINE
